// TIA Portal project "Elevator (Advanced)" (V17)

(* hardware
DEVICE "S7-1500/ET200MP station_1"  S7-1500 station
   slot 0: "Rail_0"  Rack  6ES7 590-1***0-0AA0
   slot 1: "PLC_1"  CPU 1511-1 PN  6ES7 511-1AK02-0AB0  V2.9
      slot 3: "CPU display_1"  6ES7591-1AA00-0AA0
      slot 32768: "PROFINET interface_1"  X1
         slot 32769: "Port_1"  X1 P1
         slot 32770: "Port_2"  X1 P2
      slot 34817: "Virtual CP interface port_1"  Virtual CP interface port  Virtual CP interface port
   slot 2: "DI 32x24VDC BA_1"  DI 32x24VDC BA  6ES7 521-1BL10-0AA0  V1.1
   slot 3: "DQ 32x24VDC/0.5A BA_1"  DQ 32x24VDC/0.5A BA  6ES7 522-1BL10-0AA0  V1.1
   slot 4: "AI 4xU/I/RTD/TC ST_1"  AI 4xU/I/RTD/TC ST  6ES7 531-7QD00-0AB0  V1.0
   slot 5: "AQ 4xU/I ST_1"  AQ 4xU/I ST  6ES7 532-5HD00-0AB0  V2.2
*)

// ===== PLC "PLC_1"  CPU 1511-1 PN =====

VAR_GLOBAL   // PLC tag table "IO"
   "At 1" AT %I0.0 : Bool;
   "At 2" AT %I0.1 : Bool;
   "At 3" AT %I0.2 : Bool;
   "At elevator" AT %I0.3 : Bool;
   "At entry" AT %I0.4 : Bool;
   "At exit" AT %I0.5 : Bool;
   "At 0 (low)" AT %I0.6 : Bool;
   "At 0 (high)" AT %I0.7 : Bool;
   "At 1 (low)" AT %I1.0 : Bool;
   "At 1 (high)" AT %I1.1 : Bool;
   "At 2 (low)" AT %I1.2 : Bool;
   "At 2 (high)" AT %I1.3 : Bool;
   "At 3 (low)" AT %I1.4 : Bool;
   "At 3 (high)" AT %I1.5 : Bool;
   "Start" AT %I1.6 : Bool;
   "Reset" AT %I1.7 : Bool;
   "Stop" AT %I2.0 : Bool;
   "Emergency stop" AT %I2.1 : Bool;
   "Auto" AT %I2.2 : Bool;
   "FACTORY I/O (Running)" AT %I2.3 : Bool;
   "Conveyor 0" AT %Q0.0 : Bool;
   "Conveyor 1" AT %Q0.1 : Bool;
   "Conveyor 2" AT %Q0.2 : Bool;
   "Conveyor 3" AT %Q0.3 : Bool;
   "Exit conveyor" AT %Q0.4 : Bool;
   "Load" AT %Q0.5 : Bool;
   "Unload" AT %Q0.6 : Bool;
   "Up" AT %Q0.7 : Bool;
   "Down" AT %Q1.0 : Bool;
   "Slow" AT %Q1.1 : Bool;
   "Warning light" AT %Q1.2 : Bool;
   "Start light" AT %Q1.3 : Bool;
   "Reset light" AT %Q1.4 : Bool;
   "Stop light" AT %Q1.5 : Bool;
   "Floor 1" AT %Q3.2 : Bool;
   "Floor 2" AT %Q3.3 : Bool;
   "Floor 3" AT %Q3.4 : Bool;
   "Green 1" AT %Q2.1 : Bool;
   "Yellow 1" AT %Q2.2 : Bool;
   "Red 1" AT %Q2.3 : Bool;
   "Green 2" AT %Q2.4 : Bool;
   "Yellow 2" AT %Q2.5 : Bool;
   "Red 2" AT %Q2.6 : Bool;
   "Green 3" AT %Q2.7 : Bool;
   "Yellow 3" AT %Q3.0 : Bool;
   "Red 3" AT %Q3.1 : Bool;
   "Display" AT %QW30 : Int;
END_VAR

DATA_BLOCK "HMI_Data"   // DB1
{ S7_Optimized_Access := 'TRUE' }
VERSION : 0.1
   VAR
      Start : Bool;
      Stop : Bool;
      Reset : Bool;
      Flanker : Struct
         Flank1 : Bool;
         Flank2 : Bool;
         Flank3 : Bool;
         Flank4 : Bool;
         Flank5 : Bool;
         Flank6 : Bool;
         Flank7 : Bool;
         Flank8 : Bool;
         Flank9 : Bool;
         Flank10 : Bool;
         Flank11 : Bool;
         Flank12 : Bool;
         Flank13 : Bool;
         Flank14 : Bool;
         Flank15 : Bool;
         Flank16 : Bool;
      END_STRUCT;
      Sekvensord : Int;
   END_VAR
BEGIN
END_DATA_BLOCK

// folder: System blocks/Program resources

DATA_BLOCK "IEC_Timer_0_DB"   // DB2
{ S7_Optimized_Access := 'TRUE' }
AUTHOR : Simatic
FAMILY : IEC
NAME : IEC_TMR
VERSION : 1.0
// stored: InstanceOfName IEC_TIMER
"IEC_TIMER"
BEGIN
END_DATA_BLOCK

DATA_BLOCK "IEC_Timer_1_DB"   // DB3
{ S7_Optimized_Access := 'TRUE' }
AUTHOR : Simatic
FAMILY : IEC
NAME : IEC_TMR
VERSION : 1.0
// stored: InstanceOfName IEC_TIMER
"IEC_TIMER"
BEGIN
END_DATA_BLOCK

DATA_BLOCK "IEC_Timer_2_DB"   // DB4
{ S7_Optimized_Access := 'TRUE' }
AUTHOR : Simatic
FAMILY : IEC
NAME : IEC_TMR
VERSION : 1.0
// stored: InstanceOfName IEC_TIMER
"IEC_TIMER"
BEGIN
END_DATA_BLOCK

DATA_BLOCK "IEC_Timer_3_DB"   // DB5
{ S7_Optimized_Access := 'TRUE' }
AUTHOR : Simatic
FAMILY : IEC
NAME : IEC_TMR
VERSION : 1.0
// stored: InstanceOfName IEC_TIMER
"IEC_TIMER"
BEGIN
END_DATA_BLOCK

DATA_BLOCK "IEC_Timer_4_DB"   // DB6
{ S7_Optimized_Access := 'TRUE' }
AUTHOR : Simatic
FAMILY : IEC
NAME : IEC_TMR
VERSION : 1.0
// stored: InstanceOfName IEC_TIMER
"IEC_TIMER"
BEGIN
END_DATA_BLOCK

DATA_BLOCK "IEC_Timer_5_DB"   // DB7
{ S7_Optimized_Access := 'TRUE' }
AUTHOR : Simatic
FAMILY : IEC
NAME : IEC_TMR
VERSION : 1.0
// stored: InstanceOfName IEC_TIMER
"IEC_TIMER"
BEGIN
END_DATA_BLOCK

DATA_BLOCK "IEC_Timer_6_DB"   // DB8
{ S7_Optimized_Access := 'TRUE' }
AUTHOR : Simatic
FAMILY : IEC
NAME : IEC_TMR
VERSION : 1.0
// stored: InstanceOfName IEC_TIMER
"IEC_TIMER"
BEGIN
END_DATA_BLOCK

// folder: (top level)

FUNCTION "Elevator Advanced" : Void   // FC1, LAD
{ S7_Optimized_Access := 'TRUE' }
VERSION : 0.1
   VAR_TEMP   // added for the SCL form of the ladder/FBD networks
      _w1 : Bool;
   END_VAR
BEGIN

REGION Network 1: Set Remover
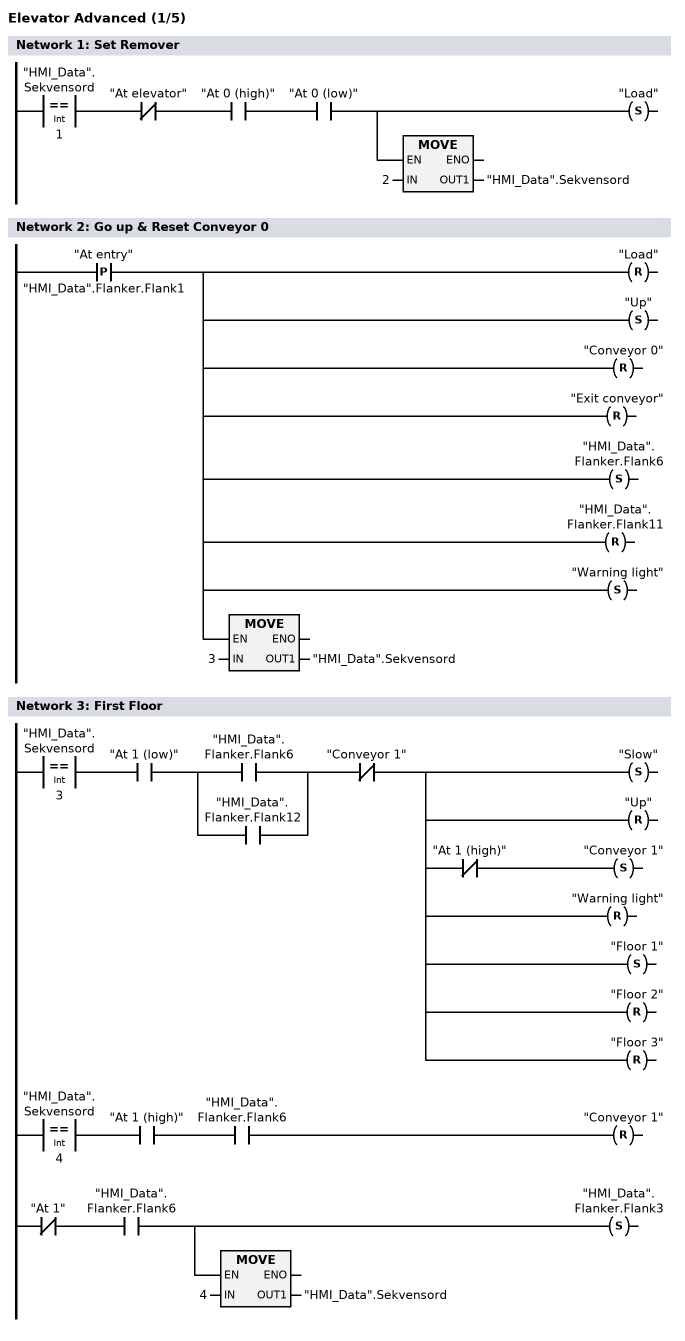
   RUNG wire#powerrail
      { S7_Templates := "SrcType := Int" } EQ_Contact(in1 := "HMI_Data".Sekvensord, in2 := 1)
      I_Contact( "At elevator" )
      Contact( "At 0 (high)" )
      Contact( "At 0 (low)" )
      wire#w1
      S_Coil( "Load" )
   END_RUNG
   RUNG wire#w1
      Move(in := 2, out1 => "HMI_Data".Sekvensord)
   END_RUNG
   // the same network as SCL:
   IF ("HMI_Data".Sekvensord = 1) AND NOT "At elevator" AND "At 0 (high)" AND "At 0 (low)" THEN
       "Load" := TRUE;
       "HMI_Data".Sekvensord := 2;
   END_IF;
END_REGION

REGION Network 2: Go up & Reset Conveyor 0
   RUNG wire#powerrail
      P_Contact(operand := "At entry", bit := "HMI_Data".Flanker.Flank1)
      wire#w1
      R_Coil( "Load" )
   END_RUNG
   RUNG wire#w1
      S_Coil( "Up" )
   END_RUNG
   RUNG wire#w1
      R_Coil( "Conveyor 0" )
   END_RUNG
   RUNG wire#w1
      R_Coil( "Exit conveyor" )
   END_RUNG
   RUNG wire#w1
      S_Coil( "HMI_Data".Flanker.Flank6 )
   END_RUNG
   RUNG wire#w1
      R_Coil( "HMI_Data".Flanker.Flank11 )
   END_RUNG
   RUNG wire#w1
      S_Coil( "Warning light" )
   END_RUNG
   RUNG wire#w1
      Move(in := 3, out1 => "HMI_Data".Sekvensord)
   END_RUNG
   // the same network as SCL:
   #_w1 := "At entry" AND NOT "HMI_Data".Flanker.Flank1;   // rising edge of "At entry"
   "HMI_Data".Flanker.Flank1 := "At entry";
   IF #_w1 THEN
       "Load" := FALSE;
       "Up" := TRUE;
       "Conveyor 0" := FALSE;
       "Exit conveyor" := FALSE;
       "HMI_Data".Flanker.Flank6 := TRUE;
       "HMI_Data".Flanker.Flank11 := FALSE;
       "Warning light" := TRUE;
       "HMI_Data".Sekvensord := 3;
   END_IF;
END_REGION

REGION Network 3: First Floor
   RUNG wire#powerrail
      { S7_Templates := "SrcType := Int" } EQ_Contact(in1 := "HMI_Data".Sekvensord, in2 := 3)
      Contact( "At 1 (low)" )
      wire#w1
      Contact( "HMI_Data".Flanker.Flank6 )
      wire#w2
      I_Contact( "Conveyor 1" )
      wire#w3
      S_Coil( "Slow" )
   END_RUNG
   RUNG wire#w1
      Contact( "HMI_Data".Flanker.Flank12 )
   END_RUNG wire#w2
   RUNG wire#w3
      R_Coil( "Up" )
   END_RUNG
   RUNG wire#w3
      I_Contact( "At 1 (high)" )
      S_Coil( "Conveyor 1" )
   END_RUNG
   RUNG wire#w3
      R_Coil( "Warning light" )
   END_RUNG
   RUNG wire#w3
      S_Coil( "Floor 1" )
   END_RUNG
   RUNG wire#w3
      R_Coil( "Floor 2" )
   END_RUNG
   RUNG wire#w3
      R_Coil( "Floor 3" )
   END_RUNG
   RUNG wire#powerrail
      { S7_Templates := "SrcType := Int" } EQ_Contact(in1 := "HMI_Data".Sekvensord, in2 := 4)
      Contact( "At 1 (high)" )
      Contact( "HMI_Data".Flanker.Flank6 )
      R_Coil( "Conveyor 1" )
   END_RUNG
   RUNG wire#powerrail
      I_Contact( "At 1" )
      Contact( "HMI_Data".Flanker.Flank6 )
      wire#w4
      S_Coil( "HMI_Data".Flanker.Flank3 )
   END_RUNG
   RUNG wire#w4
      Move(in := 4, out1 => "HMI_Data".Sekvensord)
   END_RUNG
   // the same network as SCL:
   #_w1 := ("HMI_Data".Sekvensord = 3) AND "At 1 (low)" AND ("HMI_Data".Flanker.Flank6 OR "HMI_Data".Flanker.Flank12) AND NOT "Conveyor 1";
   IF #_w1 THEN
       "Slow" := TRUE;
       "Up" := FALSE;
   END_IF;
   IF #_w1 AND NOT "At 1 (high)" THEN "Conveyor 1" := TRUE; END_IF;
   IF #_w1 THEN
       "Warning light" := FALSE;
       "Floor 1" := TRUE;
       "Floor 2" := FALSE;
       "Floor 3" := FALSE;
   END_IF;
   IF ("HMI_Data".Sekvensord = 4) AND "At 1 (high)" AND "HMI_Data".Flanker.Flank6 THEN
       "Conveyor 1" := FALSE;
   END_IF;
   IF NOT "At 1" AND "HMI_Data".Flanker.Flank6 THEN
       "HMI_Data".Flanker.Flank3 := TRUE;
       "HMI_Data".Sekvensord := 4;
   END_IF;
END_REGION

REGION Network 4: Go up & Reset Conveyor 1
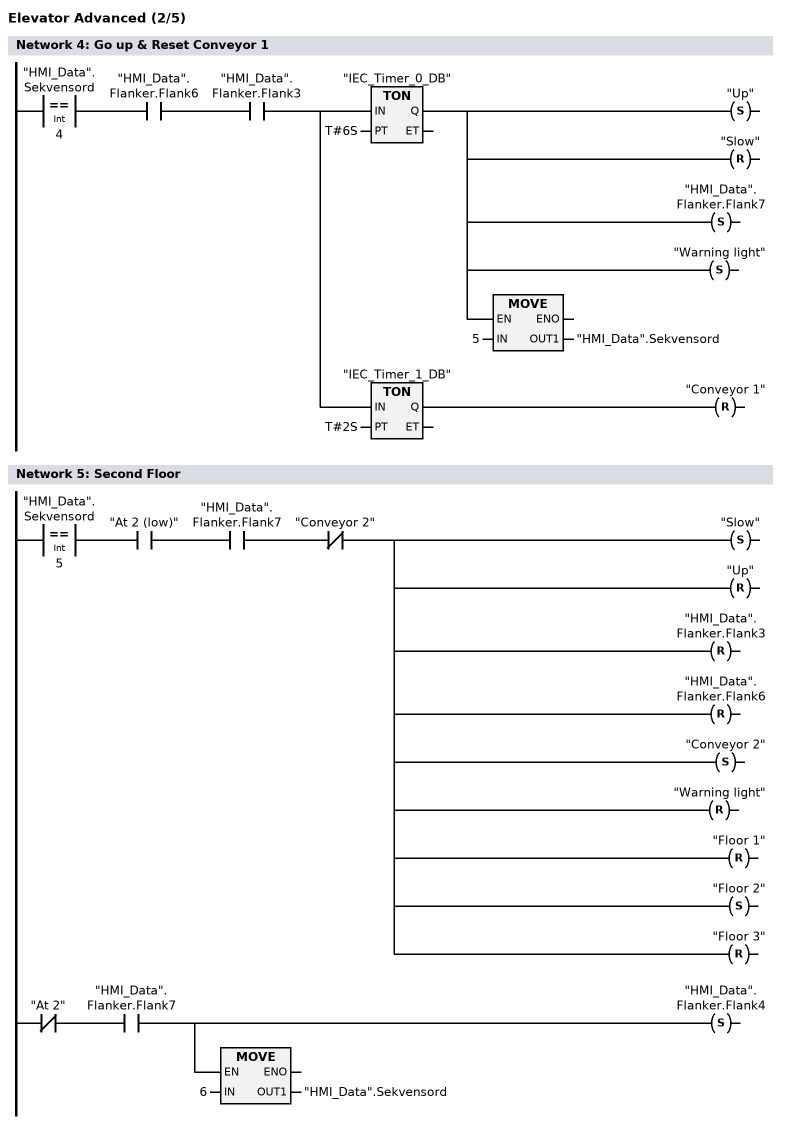
   #_w1 := ("HMI_Data".Sekvensord = 4) AND "HMI_Data".Flanker.Flank6 AND "HMI_Data".Flanker.Flank3;
   "IEC_Timer_0_DB".TON(IN := #_w1, PT := T#6S);
   IF "IEC_Timer_0_DB".Q THEN
       "Up" := TRUE;
       "Slow" := FALSE;
       "HMI_Data".Flanker.Flank7 := TRUE;
       "Warning light" := TRUE;
       "HMI_Data".Sekvensord := 5;
   END_IF;
   "IEC_Timer_1_DB".TON(IN := #_w1, PT := T#2S);
   IF "IEC_Timer_1_DB".Q THEN "Conveyor 1" := FALSE; END_IF;
END_REGION

REGION Network 5: Second Floor
   RUNG wire#powerrail
      { S7_Templates := "SrcType := Int" } EQ_Contact(in1 := "HMI_Data".Sekvensord, in2 := 5)
      Contact( "At 2 (low)" )
      Contact( "HMI_Data".Flanker.Flank7 )
      I_Contact( "Conveyor 2" )
      wire#w1
      S_Coil( "Slow" )
   END_RUNG
   RUNG wire#w1
      R_Coil( "Up" )
   END_RUNG
   RUNG wire#w1
      R_Coil( "HMI_Data".Flanker.Flank3 )
   END_RUNG
   RUNG wire#w1
      R_Coil( "HMI_Data".Flanker.Flank6 )
   END_RUNG
   RUNG wire#w1
      S_Coil( "Conveyor 2" )
   END_RUNG
   RUNG wire#w1
      R_Coil( "Warning light" )
   END_RUNG
   RUNG wire#w1
      R_Coil( "Floor 1" )
   END_RUNG
   RUNG wire#w1
      S_Coil( "Floor 2" )
   END_RUNG
   RUNG wire#w1
      R_Coil( "Floor 3" )
   END_RUNG
   RUNG wire#powerrail
      I_Contact( "At 2" )
      Contact( "HMI_Data".Flanker.Flank7 )
      wire#w2
      S_Coil( "HMI_Data".Flanker.Flank4 )
   END_RUNG
   RUNG wire#w2
      Move(in := 6, out1 => "HMI_Data".Sekvensord)
   END_RUNG
   // the same network as SCL:
   IF ("HMI_Data".Sekvensord = 5) AND "At 2 (low)" AND "HMI_Data".Flanker.Flank7 AND NOT "Conveyor 2" THEN
       "Slow" := TRUE;
       "Up" := FALSE;
       "HMI_Data".Flanker.Flank3 := FALSE;
       "HMI_Data".Flanker.Flank6 := FALSE;
   END_IF;
   #_w1 := ("HMI_Data".Sekvensord = 5) AND "At 2 (low)" AND "HMI_Data".Flanker.Flank7 AND NOT "Conveyor 2";
   IF #_w1 THEN
       "Conveyor 2" := TRUE;
       "Warning light" := FALSE;
       "Floor 1" := FALSE;
       "Floor 2" := TRUE;
       "Floor 3" := FALSE;
   END_IF;
   IF NOT "At 2" AND "HMI_Data".Flanker.Flank7 THEN
       "HMI_Data".Flanker.Flank4 := TRUE;
       "HMI_Data".Sekvensord := 6;
   END_IF;
END_REGION

REGION Network 6: Go up & Reset Conveyor 2
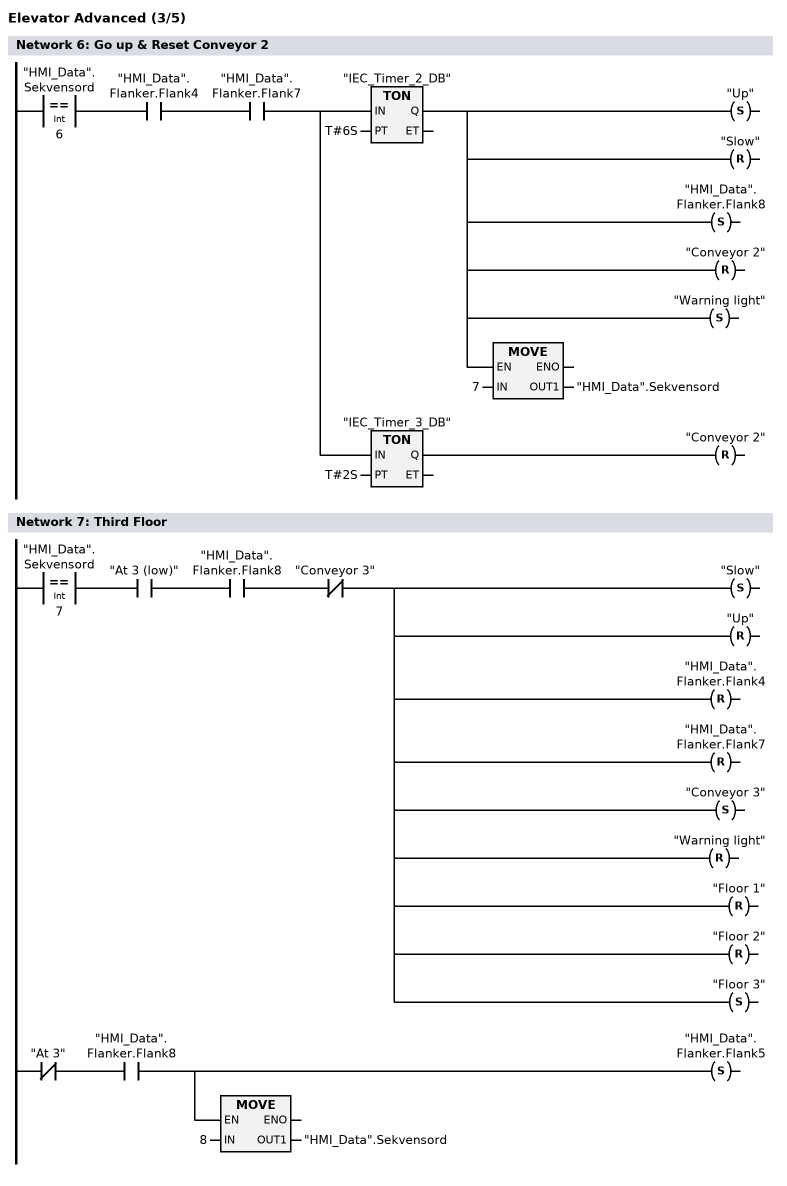
   #_w1 := ("HMI_Data".Sekvensord = 6) AND "HMI_Data".Flanker.Flank4 AND "HMI_Data".Flanker.Flank7;
   "IEC_Timer_2_DB".TON(IN := #_w1, PT := T#6S);
   IF "IEC_Timer_2_DB".Q THEN
       "Up" := TRUE;
       "Slow" := FALSE;
       "HMI_Data".Flanker.Flank8 := TRUE;
       "Conveyor 2" := FALSE;
       "Warning light" := TRUE;
       "HMI_Data".Sekvensord := 7;
   END_IF;
   "IEC_Timer_3_DB".TON(IN := #_w1, PT := T#2S);
   IF "IEC_Timer_3_DB".Q THEN "Conveyor 2" := FALSE; END_IF;
END_REGION

REGION Network 7: Third Floor
   RUNG wire#powerrail
      { S7_Templates := "SrcType := Int" } EQ_Contact(in1 := "HMI_Data".Sekvensord, in2 := 7)
      Contact( "At 3 (low)" )
      Contact( "HMI_Data".Flanker.Flank8 )
      I_Contact( "Conveyor 3" )
      wire#w1
      S_Coil( "Slow" )
   END_RUNG
   RUNG wire#w1
      R_Coil( "Up" )
   END_RUNG
   RUNG wire#w1
      R_Coil( "HMI_Data".Flanker.Flank4 )
   END_RUNG
   RUNG wire#w1
      R_Coil( "HMI_Data".Flanker.Flank7 )
   END_RUNG
   RUNG wire#w1
      S_Coil( "Conveyor 3" )
   END_RUNG
   RUNG wire#w1
      R_Coil( "Warning light" )
   END_RUNG
   RUNG wire#w1
      R_Coil( "Floor 1" )
   END_RUNG
   RUNG wire#w1
      R_Coil( "Floor 2" )
   END_RUNG
   RUNG wire#w1
      S_Coil( "Floor 3" )
   END_RUNG
   RUNG wire#powerrail
      I_Contact( "At 3" )
      Contact( "HMI_Data".Flanker.Flank8 )
      wire#w2
      S_Coil( "HMI_Data".Flanker.Flank5 )
   END_RUNG
   RUNG wire#w2
      Move(in := 8, out1 => "HMI_Data".Sekvensord)
   END_RUNG
   // the same network as SCL:
   IF ("HMI_Data".Sekvensord = 7) AND "At 3 (low)" AND "HMI_Data".Flanker.Flank8 AND NOT "Conveyor 3" THEN
       "Slow" := TRUE;
       "Up" := FALSE;
       "HMI_Data".Flanker.Flank4 := FALSE;
       "HMI_Data".Flanker.Flank7 := FALSE;
   END_IF;
   #_w1 := ("HMI_Data".Sekvensord = 7) AND "At 3 (low)" AND "HMI_Data".Flanker.Flank8 AND NOT "Conveyor 3";
   IF #_w1 THEN
       "Conveyor 3" := TRUE;
       "Warning light" := FALSE;
       "Floor 1" := FALSE;
       "Floor 2" := FALSE;
       "Floor 3" := TRUE;
   END_IF;
   IF NOT "At 3" AND "HMI_Data".Flanker.Flank8 THEN
       "HMI_Data".Flanker.Flank5 := TRUE;
       "HMI_Data".Sekvensord := 8;
   END_IF;
END_REGION

REGION Network 8: Go Down & reset Conveyor 3
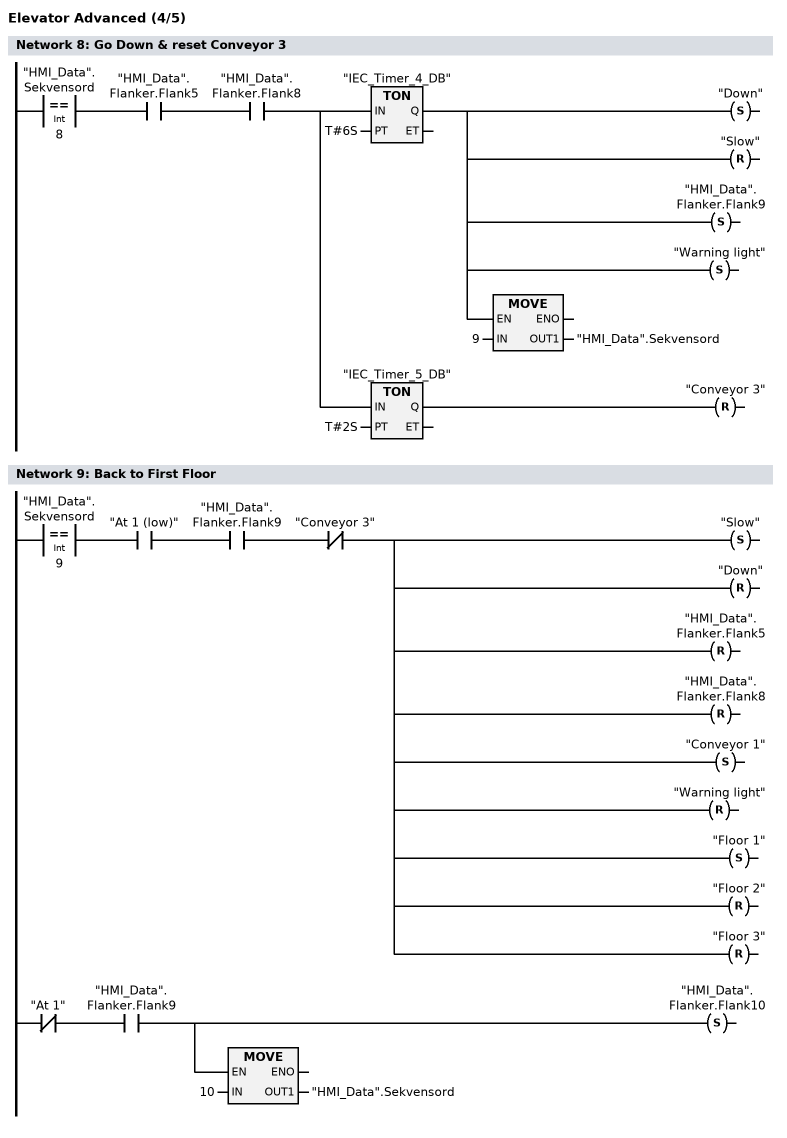
   #_w1 := ("HMI_Data".Sekvensord = 8) AND "HMI_Data".Flanker.Flank5 AND "HMI_Data".Flanker.Flank8;
   "IEC_Timer_4_DB".TON(IN := #_w1, PT := T#6S);
   IF "IEC_Timer_4_DB".Q THEN
       "Down" := TRUE;
       "Slow" := FALSE;
       "HMI_Data".Flanker.Flank9 := TRUE;
       "Warning light" := TRUE;
       "HMI_Data".Sekvensord := 9;
   END_IF;
   "IEC_Timer_5_DB".TON(IN := #_w1, PT := T#2S);
   IF "IEC_Timer_5_DB".Q THEN "Conveyor 3" := FALSE; END_IF;
END_REGION

REGION Network 9: Back to First Floor
   RUNG wire#powerrail
      { S7_Templates := "SrcType := Int" } EQ_Contact(in1 := "HMI_Data".Sekvensord, in2 := 9)
      Contact( "At 1 (low)" )
      Contact( "HMI_Data".Flanker.Flank9 )
      I_Contact( "Conveyor 3" )
      wire#w1
      S_Coil( "Slow" )
   END_RUNG
   RUNG wire#w1
      R_Coil( "Down" )
   END_RUNG
   RUNG wire#w1
      R_Coil( "HMI_Data".Flanker.Flank5 )
   END_RUNG
   RUNG wire#w1
      R_Coil( "HMI_Data".Flanker.Flank8 )
   END_RUNG
   RUNG wire#w1
      S_Coil( "Conveyor 1" )
   END_RUNG
   RUNG wire#w1
      R_Coil( "Warning light" )
   END_RUNG
   RUNG wire#w1
      S_Coil( "Floor 1" )
   END_RUNG
   RUNG wire#w1
      R_Coil( "Floor 2" )
   END_RUNG
   RUNG wire#w1
      R_Coil( "Floor 3" )
   END_RUNG
   RUNG wire#powerrail
      I_Contact( "At 1" )
      Contact( "HMI_Data".Flanker.Flank9 )
      wire#w2
      S_Coil( "HMI_Data".Flanker.Flank10 )
   END_RUNG
   RUNG wire#w2
      Move(in := 10, out1 => "HMI_Data".Sekvensord)
   END_RUNG
   // the same network as SCL:
   IF ("HMI_Data".Sekvensord = 9) AND "At 1 (low)" AND "HMI_Data".Flanker.Flank9 AND NOT "Conveyor 3" THEN
       "Slow" := TRUE;
       "Down" := FALSE;
       "HMI_Data".Flanker.Flank5 := FALSE;
       "HMI_Data".Flanker.Flank8 := FALSE;
       "Conveyor 1" := TRUE;
       "Warning light" := FALSE;
       "Floor 1" := TRUE;
       "Floor 2" := FALSE;
       "Floor 3" := FALSE;
   END_IF;
   IF NOT "At 1" AND "HMI_Data".Flanker.Flank9 THEN
       "HMI_Data".Flanker.Flank10 := TRUE;
       "HMI_Data".Sekvensord := 10;
   END_IF;
END_REGION

REGION Network 10: Floor 0
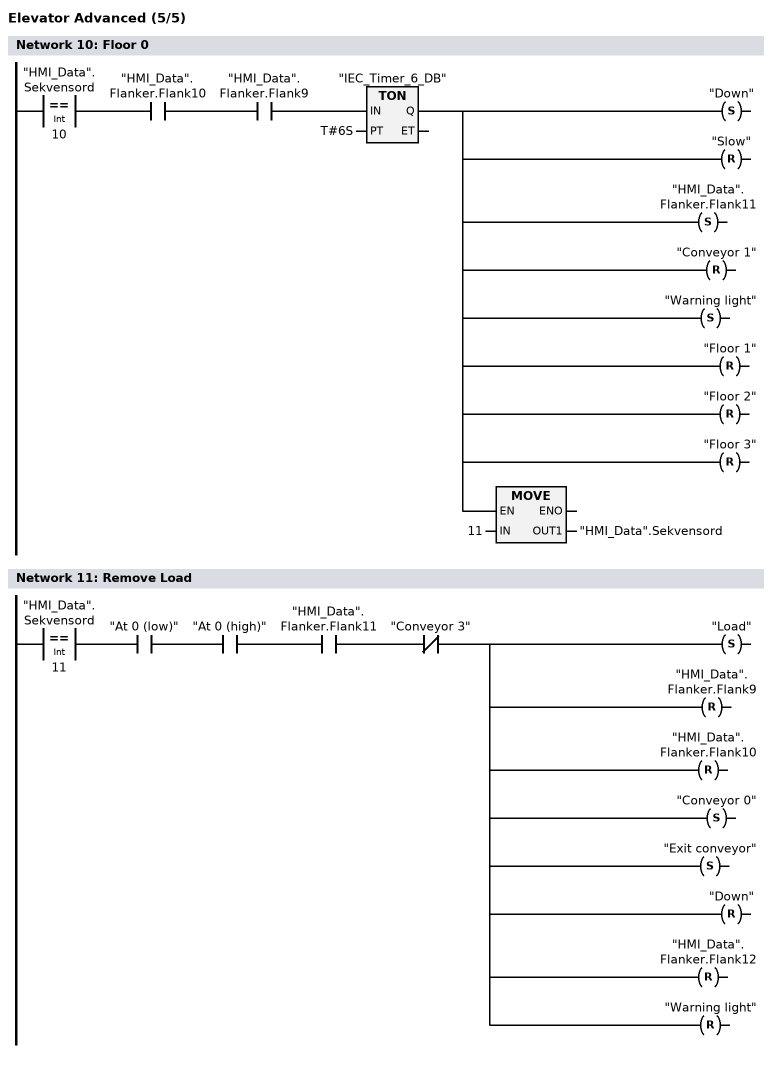
   "IEC_Timer_6_DB".TON(IN := ("HMI_Data".Sekvensord = 10) AND "HMI_Data".Flanker.Flank10 AND "HMI_Data".Flanker.Flank9,
                        PT := T#6S);
   IF "IEC_Timer_6_DB".Q THEN
       "Down" := TRUE;
       "Slow" := FALSE;
       "HMI_Data".Flanker.Flank11 := TRUE;
       "Conveyor 1" := FALSE;
       "Warning light" := TRUE;
       "Floor 1" := FALSE;
       "Floor 2" := FALSE;
       "Floor 3" := FALSE;
       "HMI_Data".Sekvensord := 11;
   END_IF;
END_REGION

REGION Network 11: Remove Load
   RUNG wire#powerrail
      { S7_Templates := "SrcType := Int" } EQ_Contact(in1 := "HMI_Data".Sekvensord, in2 := 11)
      Contact( "At 0 (low)" )
      Contact( "At 0 (high)" )
      Contact( "HMI_Data".Flanker.Flank11 )
      I_Contact( "Conveyor 3" )
      wire#w1
      S_Coil( "Load" )
   END_RUNG
   RUNG wire#w1
      R_Coil( "HMI_Data".Flanker.Flank9 )
   END_RUNG
   RUNG wire#w1
      R_Coil( "HMI_Data".Flanker.Flank10 )
   END_RUNG
   RUNG wire#w1
      S_Coil( "Conveyor 0" )
   END_RUNG
   RUNG wire#w1
      S_Coil( "Exit conveyor" )
   END_RUNG
   RUNG wire#w1
      R_Coil( "Down" )
   END_RUNG
   RUNG wire#w1
      R_Coil( "HMI_Data".Flanker.Flank12 )
   END_RUNG
   RUNG wire#w1
      R_Coil( "Warning light" )
   END_RUNG
   // the same network as SCL:
   IF ("HMI_Data".Sekvensord = 11) AND "At 0 (low)" AND "At 0 (high)" AND "HMI_Data".Flanker.Flank11 AND NOT "Conveyor 3" THEN
       "Load" := TRUE;
       "HMI_Data".Flanker.Flank9 := FALSE;
       "HMI_Data".Flanker.Flank10 := FALSE;
       "Conveyor 0" := TRUE;
       "Exit conveyor" := TRUE;
       "Down" := FALSE;
       "HMI_Data".Flanker.Flank12 := FALSE;
       "Warning light" := FALSE;
   END_IF;
END_REGION
END_FUNCTION

FUNCTION "Kör programmet" : Void   // FC2, LAD
{ S7_Optimized_Access := 'TRUE' }
VERSION : 0.1
BEGIN

REGION Network 1: Start
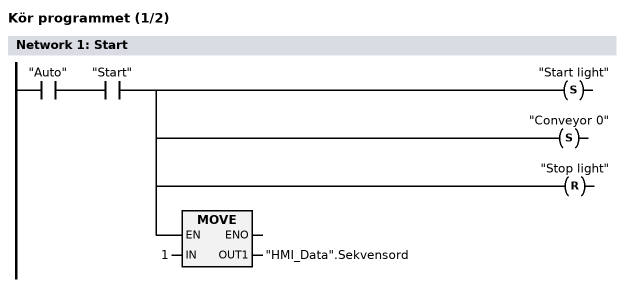
   RUNG wire#powerrail
      Contact( "Auto" )
      Contact( "Start" )
      wire#w1
      S_Coil( "Start light" )
   END_RUNG
   RUNG wire#w1
      S_Coil( "Conveyor 0" )
   END_RUNG
   RUNG wire#w1
      R_Coil( "Stop light" )
   END_RUNG
   RUNG wire#w1
      Move(in := 1, out1 => "HMI_Data".Sekvensord)
   END_RUNG
   // the same network as SCL:
   IF "Auto" AND "Start" THEN
       "Start light" := TRUE;
       "Conveyor 0" := TRUE;
       "Stop light" := FALSE;
       "HMI_Data".Sekvensord := 1;
   END_IF;
END_REGION

REGION Network 2: Reset
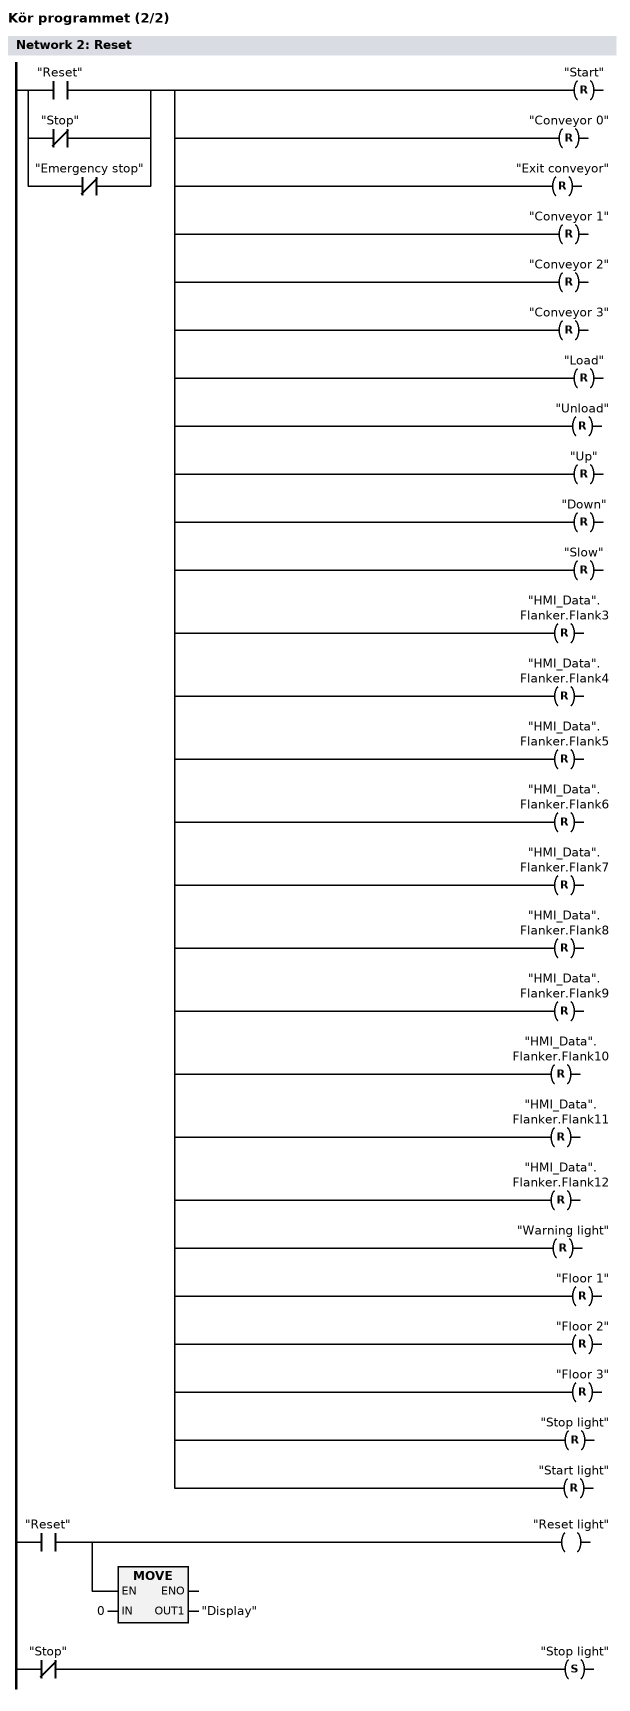
   RUNG wire#powerrail
      Contact( "Reset" )
      wire#w1
      R_Coil( "Start" )
   END_RUNG
   RUNG wire#powerrail
      I_Contact( "Stop" )
   END_RUNG wire#w1
   RUNG wire#powerrail
      I_Contact( "Emergency stop" )
   END_RUNG wire#w1
   RUNG wire#w1
      R_Coil( "Conveyor 0" )
   END_RUNG
   RUNG wire#w1
      R_Coil( "Exit conveyor" )
   END_RUNG
   RUNG wire#w1
      R_Coil( "Conveyor 1" )
   END_RUNG
   RUNG wire#w1
      R_Coil( "Conveyor 2" )
   END_RUNG
   RUNG wire#w1
      R_Coil( "Conveyor 3" )
   END_RUNG
   RUNG wire#w1
      R_Coil( "Load" )
   END_RUNG
   RUNG wire#w1
      R_Coil( "Unload" )
   END_RUNG
   RUNG wire#w1
      R_Coil( "Up" )
   END_RUNG
   RUNG wire#w1
      R_Coil( "Down" )
   END_RUNG
   RUNG wire#w1
      R_Coil( "Slow" )
   END_RUNG
   RUNG wire#w1
      R_Coil( "HMI_Data".Flanker.Flank3 )
   END_RUNG
   RUNG wire#w1
      R_Coil( "HMI_Data".Flanker.Flank4 )
   END_RUNG
   RUNG wire#w1
      R_Coil( "HMI_Data".Flanker.Flank5 )
   END_RUNG
   RUNG wire#w1
      R_Coil( "HMI_Data".Flanker.Flank6 )
   END_RUNG
   RUNG wire#w1
      R_Coil( "HMI_Data".Flanker.Flank7 )
   END_RUNG
   RUNG wire#w1
      R_Coil( "HMI_Data".Flanker.Flank8 )
   END_RUNG
   RUNG wire#w1
      R_Coil( "HMI_Data".Flanker.Flank9 )
   END_RUNG
   RUNG wire#w1
      R_Coil( "HMI_Data".Flanker.Flank10 )
   END_RUNG
   RUNG wire#w1
      R_Coil( "HMI_Data".Flanker.Flank11 )
   END_RUNG
   RUNG wire#w1
      R_Coil( "HMI_Data".Flanker.Flank12 )
   END_RUNG
   RUNG wire#w1
      R_Coil( "Warning light" )
   END_RUNG
   RUNG wire#w1
      R_Coil( "Floor 1" )
   END_RUNG
   RUNG wire#w1
      R_Coil( "Floor 2" )
   END_RUNG
   RUNG wire#w1
      R_Coil( "Floor 3" )
   END_RUNG
   RUNG wire#w1
      R_Coil( "Stop light" )
   END_RUNG
   RUNG wire#w1
      R_Coil( "Start light" )
   END_RUNG
   RUNG wire#powerrail
      Contact( "Reset" )
      wire#w2
      Coil( "Reset light" )
   END_RUNG
   RUNG wire#w2
      Move(in := 0, out1 => "Display")
   END_RUNG
   RUNG wire#powerrail
      I_Contact( "Stop" )
      S_Coil( "Stop light" )
   END_RUNG
   // the same network as SCL:
   IF "Reset" OR NOT "Stop" OR NOT "Emergency stop" THEN
       "Start" := FALSE;
       "Conveyor 0" := FALSE;
       "Exit conveyor" := FALSE;
       "Conveyor 1" := FALSE;
       "Conveyor 2" := FALSE;
       "Conveyor 3" := FALSE;
       "Load" := FALSE;
       "Unload" := FALSE;
       "Up" := FALSE;
       "Down" := FALSE;
       "Slow" := FALSE;
       "HMI_Data".Flanker.Flank3 := FALSE;
       "HMI_Data".Flanker.Flank4 := FALSE;
       "HMI_Data".Flanker.Flank5 := FALSE;
       "HMI_Data".Flanker.Flank6 := FALSE;
       "HMI_Data".Flanker.Flank7 := FALSE;
       "HMI_Data".Flanker.Flank8 := FALSE;
       "HMI_Data".Flanker.Flank9 := FALSE;
       "HMI_Data".Flanker.Flank10 := FALSE;
       "HMI_Data".Flanker.Flank11 := FALSE;
       "HMI_Data".Flanker.Flank12 := FALSE;
       "Warning light" := FALSE;
       "Floor 1" := FALSE;
       "Floor 2" := FALSE;
       "Floor 3" := FALSE;
       "Stop light" := FALSE;
       "Start light" := FALSE;
   END_IF;
   "Reset light" := "Reset";
   IF "Reset" THEN "Display" := 0; END_IF;
   IF NOT "Stop" THEN "Stop light" := TRUE; END_IF;
END_REGION
END_FUNCTION

FUNCTION "Raknare" : Void   // FC3, LAD
{ S7_Optimized_Access := 'TRUE' }
VERSION : 0.1
   VAR_TEMP   // added for the SCL form of the ladder/FBD networks
      _w1 : Bool;
   END_VAR
BEGIN

REGION Network 1: first Floor
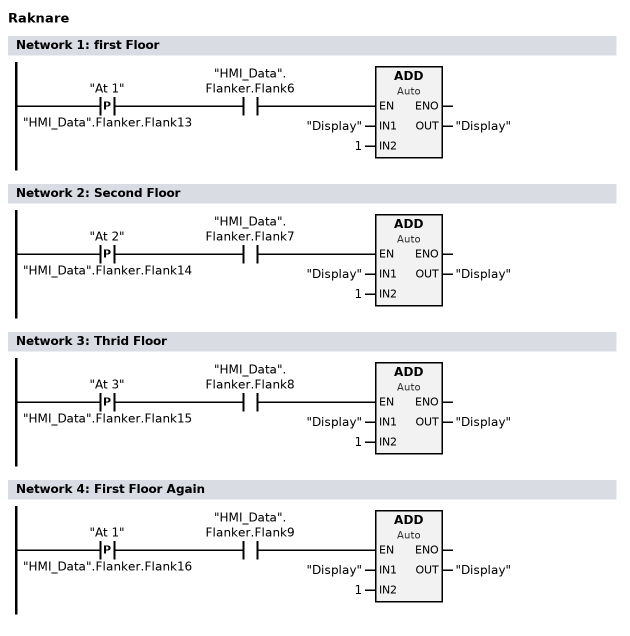
   RUNG wire#powerrail
      P_Contact(operand := "At 1", bit := "HMI_Data".Flanker.Flank13)
      Contact( "HMI_Data".Flanker.Flank6 )
      Add(in1 := "Display", in2 := 1, out => "Display")
   END_RUNG
   // the same network as SCL:
   #_w1 := "At 1" AND NOT "HMI_Data".Flanker.Flank13;   // rising edge of "At 1"
   "HMI_Data".Flanker.Flank13 := "At 1";
   IF #_w1 AND "HMI_Data".Flanker.Flank6 THEN "Display" := "Display" + 1; END_IF;
END_REGION

REGION Network 2: Second Floor
   RUNG wire#powerrail
      P_Contact(operand := "At 2", bit := "HMI_Data".Flanker.Flank14)
      Contact( "HMI_Data".Flanker.Flank7 )
      Add(in1 := "Display", in2 := 1, out => "Display")
   END_RUNG
   // the same network as SCL:
   #_w1 := "At 2" AND NOT "HMI_Data".Flanker.Flank14;   // rising edge of "At 2"
   "HMI_Data".Flanker.Flank14 := "At 2";
   IF #_w1 AND "HMI_Data".Flanker.Flank7 THEN "Display" := "Display" + 1; END_IF;
END_REGION

REGION Network 3: Thrid Floor
   RUNG wire#powerrail
      P_Contact(operand := "At 3", bit := "HMI_Data".Flanker.Flank15)
      Contact( "HMI_Data".Flanker.Flank8 )
      Add(in1 := "Display", in2 := 1, out => "Display")
   END_RUNG
   // the same network as SCL:
   #_w1 := "At 3" AND NOT "HMI_Data".Flanker.Flank15;   // rising edge of "At 3"
   "HMI_Data".Flanker.Flank15 := "At 3";
   IF #_w1 AND "HMI_Data".Flanker.Flank8 THEN "Display" := "Display" + 1; END_IF;
END_REGION

REGION Network 4: First Floor Again
   RUNG wire#powerrail
      P_Contact(operand := "At 1", bit := "HMI_Data".Flanker.Flank16)
      Contact( "HMI_Data".Flanker.Flank9 )
      Add(in1 := "Display", in2 := 1, out => "Display")
   END_RUNG
   // the same network as SCL:
   #_w1 := "At 1" AND NOT "HMI_Data".Flanker.Flank16;   // rising edge of "At 1"
   "HMI_Data".Flanker.Flank16 := "At 1";
   IF #_w1 AND "HMI_Data".Flanker.Flank9 THEN "Display" := "Display" + 1; END_IF;
END_REGION
END_FUNCTION

ORGANIZATION_BLOCK "Main"   // OB1, LAD, ProgramCycle
TITLE = "Main Program Sweep (Cycle)"
{ S7_Optimized_Access := 'TRUE' }
VERSION : 0.1
   VAR_INPUT
      Initial_Call : Bool;   // Initial call of this OB
      Remanence : Bool;   // =True, if remanent data are available
   END_VAR
BEGIN

REGION Network 1
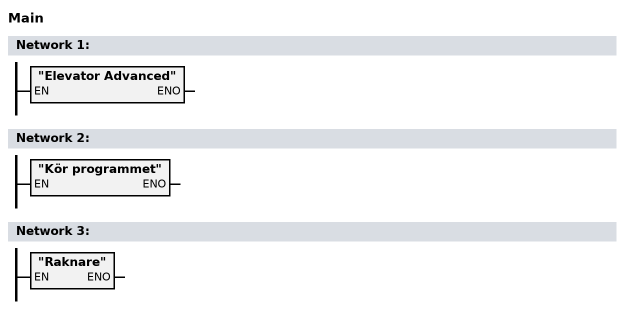
   RUNG wire#powerrail
      "Elevator Advanced"()
   END_RUNG
   // the same network as SCL:
   "Elevator Advanced"();
END_REGION

REGION Network 2
   RUNG wire#powerrail
      "Kör programmet"()
   END_RUNG
   // the same network as SCL:
   "Kör programmet"();
END_REGION

REGION Network 3
   RUNG wire#powerrail
      "Raknare"()
   END_RUNG
   // the same network as SCL:
   "Raknare"();
END_REGION
END_ORGANIZATION_BLOCK